{attribute addProperty BoxType "EL2809-0000-0018"}
{attribute addProperty Id "WcStateAT %I*BIT10.1250"}
{attribute addProperty CRC "682125173"}
{attribute addProperty SizeInBites "1"}
{attribute addProperty SizeInBytes "0.125"}
TYPE WcState_28A86775 :
STRUCT
	{attribute addProperty Name "WcState"}
	WcState AT %I* : BOOL;
END_STRUCT
END_TYPE

(* stored: Version 1.2.0.0, ProductVersion 3.1.4024.9
   DUT WcState_28A86775: Id {db819636-5123-0cf4-2897-5b4bc37604fb} *)
